ABB RobotStudio station: Calvo_Petrigh_Embolsadora_Cemento_20241123-220002.rsstn

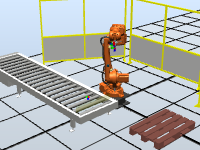
Station Calvo_Petrigh_Embolsadora_Cemento (saved by RobotStudio 6.8.8307.1040)
Controller IRB_4600_60kg_2.05m, task T_ROB1: task frame (RAPID world) sits at (0, 0, 225) mm in the station
Controller IRB_4600_60kg_2.05m
  mechanical unit ROB_1: IRB4600_60_205__02, 6 joints, base frame (0, 0, 0) mm
Layout (positions relative to the parent item):
  - IRB4600_60_205__02 [mechanism, from Robots\IRB4600_60_205__02.rslib] at (0, 0, 225) mm; joint values [-0.7854, -0.1029, -0.0935, 0, 1.7672, 3.1416] (rad or m)
  - Robotpedestal1400_H240 [part, from Equipment\Robot Pedestal 1400 H240.rslib] at (-30, 0, 0) mm
  - 950_4000_h2 [part, from Equipment\Conveyor 950 4000 h2.rslib] at (-3500, -1500, 0) mm
  - Euro Pallet [graphiccomponentgroup, from Equipment\Euro Pallet.rslib] at (1200, 450, 0) mm, rotated rx 0 ry 0 rz -90 deg
    - Body 1 [part, from Equipment\Euro Pallet.rslib]
  - BolsaCemento [part, from Libraries\BolsaCemento.rslib]
  - SmartComponent_1 [smart component]
      signals: DO CementReady
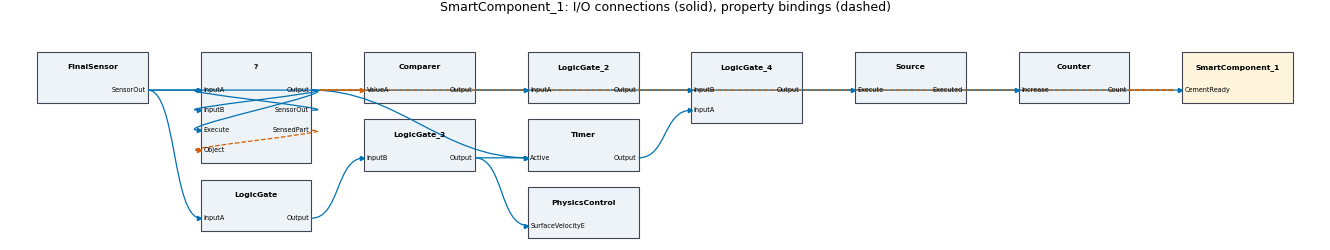
      connections:
        FinalSensor.SensorOut -> ?.InputA
        ?.Output -> Timer.Active
        ?.SensorOut -> ?.InputA
        ?.Output -> ?.InputB
        ?.Output -> ?.Execute
        FinalSensor.SensorOut -> LogicGate.InputA
        Source.Executed -> Counter.Increase
        Comparer.Output -> LogicGate_2.InputA
        LogicGate.Output -> LogicGate_3.InputB
        LogicGate_3.Output -> Timer.Active
        LogicGate_3.Output -> PhysicsControl.SurfaceVelocityEnabled
        FinalSensor.SensorOut -> SmartComponent_1.CementReady
        LogicGate_2.Output -> LogicGate_4.InputB
        Timer.Output -> LogicGate_4.InputA
        LogicGate_4.Output -> Source.Execute
        ?.SensedPart => ?.Object
        Counter.Count => Comparer.ValueA
    - Timer [smart component, from Components\Timer.rslib]
        properties: StartTime=0; Interval=3; Repeat=true; CurrentTime=0.552
    - Source [smart component, from Components\Source.rslib] at (-3343.95, -1564.26, 561.55) mm
        properties: Source=BolsaCemento; Copy=(none); Parent=(none); Position=[-3.1 -1 0.46]; Orientation=[0 0 0]; Transient=false; PhysicsBehavior=3
    - FinalSensor [smart component, from Components\PlaneSensor.rslib] at (500, -1525, 450) mm
        properties: Origin=[-0.05 0 0]; Axis1=[0 0 0.15]; Axis2=[0 0.95 0]; SensedPart=(none)
      - _sensorPart_ [part]
    - LogicGate [smart component, from Components\LogicGate.rslib]
        properties: Operator=NOT; Delay=0
    - PhysicsControl [smart component, from Components\PhysicsControl.rslib]
        properties: Object=950_4000_h2; Behavior=1; SurfaceVelocity=0.3
    - Counter [smart component, from Components\Counter.rslib]
        properties: Count=40
    - Comparer [smart component, from Components\Comparer.rslib]
        properties: ValueA=40; Operator===; ValueB=40
    - LogicGate_2 [smart component, from Components\LogicGate.rslib]
        properties: Operator=NOT; Delay=0
    - LogicGate_3 [smart component, from Components\LogicGate.rslib]
        properties: Operator=AND; Delay=0.3
    - LogicGate_4 [smart component, from Components\LogicGate.rslib]
        properties: Operator=AND; Delay=0
  - Fence_2500 [graphiccomponentgroup, from Equipment\Fence_2500.rslib] at (-3000, 0, 0) mm, rotated rx 0 ry 0 rz -30 deg
    - Body 1 [part, from Equipment\Fence_2500.rslib]
    - Body 2 [part, from Equipment\Fence_2500.rslib]
  - Fence_2500_2 [graphiccomponentgroup, from Equipment\Fence_2500.rslib] at (-1500, 2100, 0) mm, rotated rx 0 ry 0 rz -90 deg
    - Body 1 [part, from Equipment\Fence_2500.rslib]
    - Body 2 [part, from Equipment\Fence_2500.rslib]
  - Fence_740 [graphiccomponentgroup, from Equipment\Fence_740.rslib] at (1500, 1300, 0) mm, rotated rx 0 ry 0 rz 30 deg
    - Body 1 [part, from Equipment\Fence_740.rslib]
    - Body 2 [part, from Equipment\Fence_740.rslib]
  - Smart_Gripper_Servo_Fingers [mechanism, from Tools\ABB_Smart_Gripper_Servo_Fingers.rslib] at (700, -700, 1839.2) mm, rotated rx -180 ry 0 rz -45 deg; joint values [0] (rad or m)
Attachment: Smart_Gripper_Servo_Fingers is attached to IRB4600_60_205__02 / Link6
EventTableEntry 980: Group=, Trigger=PickCement 981, Actions=[EventTableActionAttach 982], Comment=, ActivationMode=2, Cyclic=false
EventTableTriggerIO 981: IOValue=[1], IRC5Controller=? -1, Operator=0, SignalSource=IRB_4600_60kg_2.05m 491
EventTableActionAttach 982: AttachmentParent=Smart_Gripper_Servo_Fingers 1179, AttachmentChild=? -1, MountObject=true, Offset=[X=1, Y=0, Z=0, W=0, X=0, Y=1, Z=0, W=0, X=0, Y=0, Z=1, W=0, X=0, Y=0, Z=0, W=1], FlangeIndext=0, FindNearest=true
EventTableEntry 983: Group=, Trigger=PickCement 984, Actions=[EventTableActionDetach 985], Comment=, ActivationMode=2, Cyclic=false
EventTableTriggerIO 984: IOValue=[0], IRC5Controller=? -1, Operator=0, SignalSource=IRB_4600_60kg_2.05m 491
EventTableActionDetach 985: AttachmentParent=Smart_Gripper_Servo_Fingers 1179, AttachmentChild=? -1
EventTableTriggerIO 1158: IOValue=[1], IRC5Controller=? -1, Operator=0, SignalSource=IRB_4600_60kg_2.05m 491
EventTableTriggerIO 1159: IOValue=[0], IRC5Controller=? -1, Operator=0, SignalSource=IRB_4600_60kg_2.05m 491
Station logic (signal -> signal, property => property):
  SmartComponent_1.CementReady -> IRB_4600_60kg_2.05m.CementReady
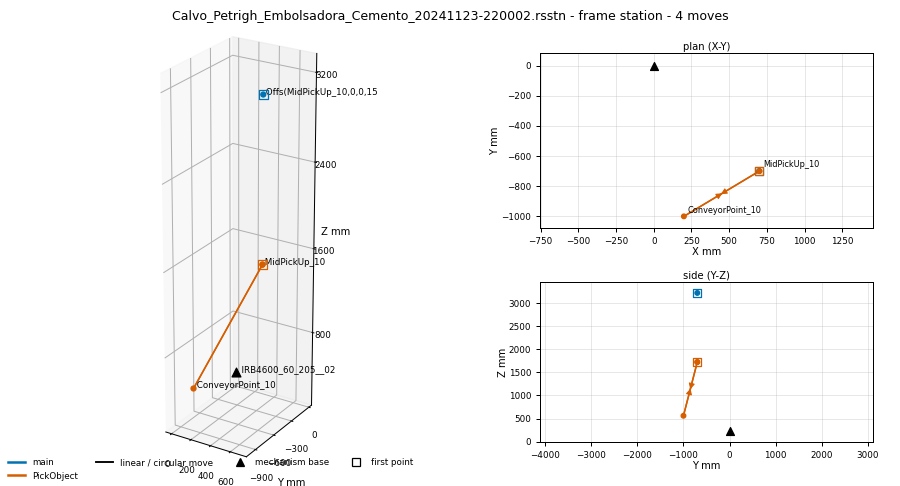
[picture p0: tool path of Calvo_Petrigh_Embolsadora_Cemento_20241123-220002.rsstn in frame station, 4 of 5 moves have a stored position in this frame; points joined in program order, loops and branches not executed]
Targets, tools, work objects and paths stored in the station, written as RAPID:
! task T_ROB1
MODULE CalibData
  PERS tooldata Servo:=[TRUE,[[0,0,114.2],[1,0,0,0]],[0.215,[8.7,12.3,49.2],[1,0,0,0],0.00021,0.00024,0.00009]];
  PERS tooldata VaccumOne:=[TRUE,[[63.5,18.5,37.5],[0.707106781,0,0.707106781,0]],[0.24,[8.2,12.5,48.1],[1,0,0,0],0.00022,0.00024,0.00009]];
  PERS tooldata Camera:=[TRUE,[[-7.3,28.3,35.1],[0.5,-0.5,0.5,0.5]],[0.24,[8.2,12.5,48.1],[1,0,0,0],0.00022,0.00024,0.00009]];
ENDMODULE

! task T_ROB1
MODULE StackCement
  CONST robtarget MidPickUp_10:=[[700,-700,1500],[0,0.923879533,-0.382683432,0],[-1,0,1,0],[9E+09,9E+09,9E+09,9E+09,9E+09,9E+09]];
  CONST robtarget ConveyorPoint_10:=[[200,-1000,335],[0,1,0,0],[-1,0,1,0],[9E+09,9E+09,9E+09,9E+09,9E+09,9E+09]];
  PROC main()
    Reset PickCement;
    WaitDI CementReady,1;
    PickObject;
    MoveL StackPositions{i},v1000,z100,Servo\WObj:=wobj0;
    DropObject;
    MoveL Offs(MidPickUp_10, 0, 0, 1500),v1000,z100,Servo\WObj:=wobj0;
  ENDPROC
  PROC PickObject()
    MoveL MidPickUp_10,v1000,z100,Servo\WObj:=wobj0;
    MoveL ConveyorPoint_10,v1000,z100,Servo\WObj:=wobj0;
    Set PickCement;
    WaitTime 0.5;
    MoveL MidPickUp_10,v1000,z100,Servo\WObj:=wobj0;
  ENDPROC
  PROC DropObject()
    WaitTime 0.5;
    Reset PickCement;
    WaitTime 0.5;
  ENDPROC
ENDMODULE

